INTERFACE I_ENGINE EXTENDS I_GENERAL_OBJECT

METHOD M_Off : BOOL
VAR_INPUT
END_VAR
END_METHOD

METHOD M_On : BOOL
VAR_INPUT
END_VAR
END_METHOD

METHOD M_SetReady : BOOL
VAR_INPUT
END_VAR
END_METHOD

PROPERTY P_Busy : BOOL
GET
END_GET
END_PROPERTY

PROPERTY P_ReadyState : BOOL
GET
END_GET
END_PROPERTY

PROPERTY P_State : BOOL
GET
END_GET
END_PROPERTY

END_INTERFACE

(* stored: Version 1.1.0.1, ProductVersion 3.1.4024.12
   Itf I_ENGINE: Id {53c66e4b-2c24-4324-807a-99a6516a1556}
   Method M_Off: Id {40151c6b-cb62-4d28-8a36-ca4eb85af945}
   Method M_On: Id {d8d76e68-4a2b-4d8c-927c-fd85975be334}
   Method M_SetReady: Id {4e8be09a-71bb-4020-a4b7-e7ef5050e1a1}
   Property P_Busy: Id {e650d9c8-c935-46ba-b63f-6ce5291ee12f}
   Get Get: Id {4c865fd4-ffd1-4df1-9af0-d873a34b375c}
   Property P_ReadyState: Id {958edc02-5bcc-4813-991b-a6103afd8def}
   Get Get: Id {0b2ed8ba-cfde-4758-9655-c7e9f6ac6ca4}
   Property P_State: Id {9368ce12-0804-41b4-abeb-930af80dc7f3}
   Get Get: Id {4cf1cb3a-87ab-4eb1-8f2e-80a02f0f3713} *)
